FUNCTION_BLOCK "EM_CIP"
{ S7_Optimized_Access := 'TRUE' }


BEGIN

END_FUNCTION_BLOCK
